{attribute 'linkalways'} 
{attribute 'no_explicit_call' := 'This FB is a CLASS and must be accessed using methods or properties'}
{attribute 'enable_dynamic_creation'}
FUNCTION_BLOCK Node_F_VN_FillContainerExp_USINT EXTENDS VisionNode
VAR
    ipContainer : _ITcVnContainer;
    nValue : _USINT(0);
    nStartIdx : _ULINT(0);
    nCount : _ULINT(0);
    hrPrev : _HRESULT(S_OK);
    hresult : _HRESULT(S_OK);
END_VAR

METHOD PUBLIC  Clone : I_Node
VAR
    pNode : POINTER TO Node_F_VN_FillContainerExp_USINT;
END_VAR
pNode := __NEW(Node_F_VN_FillContainerExp_USINT);
Clone := pNode^;
END_METHOD

METHOD FB_init : BOOL
VAR_INPUT
    bInitRetains : BOOL; // if TRUE, the retain variables are initialized (warm start / cold start)
    bInCopyCode : BOOL;  // if TRUE, the instance afterwards gets moved into the copy code (online change)
END_VAR
AddInput('ipContainer', ipContainer);
AddInput('nValue', nValue);
AddInput('nStartIdx', nStartIdx);
AddInput('nCount', nCount);
AddInput('hrPrev', hrPrev);
AddOutput('ipContainer', ipContainer);
AddOutput('hresult',hresult);
END_METHOD

METHOD PROTECTED OnExecute : HRESULT
hresult.Value := F_VN_FillContainerExp_USINT(
    ipContainer := ipContainer.Value,
    nValue := nValue.Value,
    nStartIdx := nStartIdx.Value,
    nCount := nCount.Value,
    hrPrev:= hrPrev.Value);
END_METHOD

METHOD PUBLIC PreExecutionCheck
VAR_INPUT
    Check : I_PreExecutionChecks;
END_VAR
Check.IsTrue(ipContainer.IsValid, 'ipContainer must be a valid container');
Check.IsTrue(ipContainer.HasType(TC_GLOBAL_CONST_LIST.ContainerType_Vector_USINT), 'ipContainer contains incorrect type');
END_METHOD

END_FUNCTION_BLOCK

(* stored: Version 1.1.0.1, ProductVersion 3.1.4024.13
   POU Node_F_VN_FillContainerExp_USINT: Id {14c76d5c-0f26-499a-8264-180fe03ceb50}, SpecialFunc None
   Folder Constructor: Id {09b4cf70-d903-43b2-ac37-8e2db119e3f5}
   Method Clone: Id {fc0b881f-1c2e-4975-a433-dc0fe0bf744b}
   Method FB_init: Id {3bcba92d-18fd-4b38-89d1-9f456f74a8b9}
   Method OnExecute: Id {9c8a15a5-462a-4d7a-b4a2-bdf834cb5c1d}
   Method PreExecutionCheck: Id {c811dc14-3128-42df-b06f-6d7e09fca74c} *)
